{attribute 'linkalways'} 
{attribute 'no_explicit_call' := 'This FB is a CLASS and must be accessed using methods or properties'}
{attribute 'enable_dynamic_creation'}
FUNCTION_BLOCK FINAL SUB_WORD EXTENDS Node
VAR
	in1 : _WORD(0);
	in2 : _WORD(0);
	out : _WORD(0);
END_VAR

METHOD PUBLIC Clone : I_Node
VAR
	pNode : POINTER TO SUB_WORD;
END_VAR
pNode := __NEW(SUB_WORD);
Clone := pNode^;
END_METHOD

METHOD FB_init : BOOL
VAR_INPUT
	bInitRetains : BOOL; // if TRUE, the retain variables are initialized (warm start / cold start)
	bInCopyCode : BOOL;  // if TRUE, the instance afterwards gets moved into the copy code (online change)
END_VAR
AddInput('in1',THIS^.in1);
AddInput('in2',THIS^.in2);
AddOutput('out', THIS^.out);
END_METHOD

METHOD PROTECTED OnExecute
VAR
END_VAR
out.Value := in1.Value - in2.Value;
END_METHOD

END_FUNCTION_BLOCK

(* stored: Version 1.1.0.1, ProductVersion 3.1.4024.15
   POU SUB_WORD: Id {0209d59e-4b32-49e9-bc28-4d97c52e8324}, SpecialFunc None
   Folder Constructor: Id {ed3ca907-1566-497c-88f8-4ad4aa63409e}
   Method Clone: Id {1d1702a3-a95f-4ff3-a9d1-0ba4008201b8}
   Method FB_init: Id {2105634e-518e-4f68-96ca-909930811ab1}
   Method OnExecute: Id {29400693-9686-4882-9c27-27cfa037036b} *)
